Staubli VAL3: setBitAt.pgx

public program setBitAt(num x_nByteIndex, num x_nBitIndex, bool x_bBit, num& x_nBuffer[])
begin

  if x_nBitIndex>7
    return
  endIf

 if x_bBit
    x_nBuffer[x_nByteIndex]=bOr(power(2,x_nBitIndex), x_nBuffer[x_nByteIndex])
  else
    x_nBuffer[x_nByteIndex]=bAnd(power(2,8)-power(2,x_nBitIndex)-1, x_nBuffer[x_nByteIndex])
  endIf

end
